FUNCTION_BLOCK Q_ObjHideShow (* Command Hide/Show Object (Container) ( Part 6 - F.2 ) *)
  (* Standard: ISO 11783-6; Description: Copyright (c) 2022 HR Agrartechnik GmbH This program and the accompanying materials are made available under the terms of the Eclipse Public License 2.0 which is available at https://www.eclipse.org/legal/epl-2.0/ SPDX-License-Identifier: EPL-2.0 see Description Tab *)
  (* Version 1.0, 2022-07-08, Franz Höpfinger, HR Agrartechnik GmbH *)
  PACKAGE isobus::UT::Q;
  IMPORT eclipse4diac::core::TypeHash;
  IMPORT isobus::UT::Q::IDs::ID_NULL;
  (* Documentation:
  Command Hide/Show Object (Container) ( Part 6 - F.2 )
   The Hide/Show Object command is used to hide or show a container object.
   param[in] {objectId, uint16_t}
   Object ID of Container
   param[in] {visible, bool}
   0 = Hide, 1 = Show
   Return Values: 
   int16_t
    - VT_E_NO_ERR (0) - OK
   - VT_E_OVERFLOW (-6) - buffer overflow
   - VT_E_NOACT (-8) - Command not possible in current state
   - VT_E_NO_INSTANCE (-21) - No VT client available
   - VT_E_ISO_INSTANCE_INVALID (-129) - Identifier for instance (connection) invalid
   - VT_E_HANDLE_INVALID (-128) - ErrorCause: invalid Handle
   - VT_E_NOT_ALIVE (-130) - Identifier for instance valid, but VT Dead.
  *)
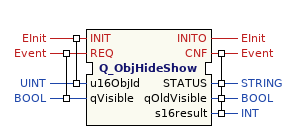
  EVENT_INPUT
    INIT : EInit WITH u16ObjId; (* Service Initialization *)
    REQ WITH qVisible; (* Service Request *)
  END_EVENT
  EVENT_OUTPUT
    INITO : EInit; (* Initialization Confirm *)
    CNF WITH STATUS, qOldVisible, s16result; (* Confirmation of Requested Service *)
  END_EVENT
  VAR_INPUT
    u16ObjId : UINT := ID_NULL; (* Object ID *)
    qVisible : BOOL; (* 0 == disable, 1 == enable *)
  END_VAR
  VAR_OUTPUT
    STATUS : STRING; (* Service Status *)
    qOldVisible : BOOL; (* Old value of Visible *)
    s16result : INT; (* retval see description *)
  END_VAR
END_FUNCTION_BLOCK
